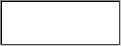
VISUALIZATION VISU_HMI_SUBSYSTEM_BUTTON  // 121x46
VAR_IN_OUT
    m_Hmi : FB_HMI_BUTTON;
END_VAR
    Rectangle (0,0 120x45), invisible if: m_Hmi.bIsNotOrange
    Rectangle (0,0 120x45), invisible if: m_Hmi.bIsNotGray
    Rectangle (0,0 120x45), invisible if: m_Hmi.bIsNotBlue
    Rectangle (0,0 120x45), invisible if: m_Hmi.bIsNotRed
    Rectangle (0,0 120x45), invisible if: m_Hmi.bIsNotGreen
    Rectangle (0,0 120x45), "%s", text variable: m_Hmi.sName
    Rectangle (0,0 120x45), invisible if: m_Hmi.bNotActivated
    Line (0,44) (120,44), invisible if: m_Hmi.bActivated
    Line (119,0) (119,45), invisible if: m_Hmi.bActivated
    Line (118,0) (0,0), invisible if: m_Hmi.bActivated
    Line (0,45) (0,0), invisible if: m_Hmi.bActivated
    Line (120,45) (120,1), invisible if: m_Hmi.bNotActivated
    Line (0,1) (119,1), invisible if: m_Hmi.bNotActivated
    Line (1,0) (1,45), invisible if: m_Hmi.bNotActivated
    Line (120,45) (1,45), invisible if: m_Hmi.bNotActivated
END_VISUALIZATION

(* stored: Version 1.1.0.1, ProductVersion 3.1.4024.14
   Visu VISU_HMI_SUBSYSTEM_BUTTON: Id {d082562c-c66c-48fd-8cf9-328019ac6a9f} *)
